FUNCTION_BLOCK PUBLIC FB_LampSetDirect
VAR
	nLightLevel			: BYTE(0..100);
END_VAR

// Sets the control value to a value between 0 and 100.
METHOD PUBLIC SetLightLevel
VAR_INPUT
	nNewLightLevel		: BYTE(0..100);
END_VAR
nLightLevel := nNewLightLevel;
END_METHOD

END_FUNCTION_BLOCK

(* stored: Version 1.1.0.1, ProductVersion 3.1.4024.9
   POU FB_LampSetDirect: Id {c9363aa1-33e3-41da-adea-7faeb59d6855}, SpecialFunc None
   Method SetLightLevel: Id {4b6fea93-5fee-4ee1-8a77-261782e46dcf} *)
